FUNCTION_BLOCK Test_TimeAsString_IncludesLeadingZeros EXTENDS TUnitTestBase
VAR
    TimeStruct : TIMESTRUCT := (wHour := 6, wMinute := 5, wSecond := 4);
END_VAR

Assertion.AssertEquals_STRING(
    Expected := '06:05:04',
    Actual   := F_TimeAsString(TimeStruct),
    ObjectName := _TestName,
    VariableName  := 'F_TimeAsString(TimeStruct)');


Test_Finished();

END_FUNCTION_BLOCK

(* stored: Version 1.1.0.1, ProductVersion 3.1.4024.3
   POU Test_TimeAsString_IncludesLeadingZeros: Id {72a01420-e5e9-02f9-2a71-637672ec7977}, SpecialFunc None *)
